// TIA Portal V19 export
TYPE "UDT_MTRFAULTS"
   STRUCT
      ctrl : Struct   // External data (Primary alarm data - alarm & plc ackn)
         alarm_ftr : Bool := false;
         alarm_fts : Bool := false;
         alarm_mcb : Bool := false;
         alarm_ctrl : Bool := false;
         alarm_vfd : Bool := false;
         alarm_il : Bool := false;
         bit14 : Bool := false;
         bit15 : Bool := false;
         plcackn_ftr : Bool := false;
         plcackn_fts : Bool := false;
         plcackn_mcb : Bool := false;
         plcackn_ctrl : Bool := false;
         plcackn_vfd : Bool := false;
         plcackn_il : Bool := false;
         bit6 : Bool := false;
         bit7 : Bool := false;
      END_STRUCT;
      status : Struct   // External data (Secondary alarm data - siren & hmi ackn)
         siren_ftr : Bool := false;
         siren_fts : Bool := false;
         siren_mcb : Bool := false;
         siren_ctrl : Bool := false;
         siren_vfd : Bool := false;
         siren_il : Bool := false;
         bit14 : Bool := false;
         bit15 : Bool := false;
         hmiackn_ftr : Bool := false;
         hmiackn_fts : Bool := false;
         hmiackn_mcb : Bool := false;
         hmiackn_ctrl : Bool := false;
         hmiackn_vfd : Bool := false;
         hmiackn_il : Bool := false;
         bit6 : Bool := false;
         bit7 : Bool := false;
      END_STRUCT;
   END_STRUCT;
END_TYPE
